PROGRAM pump_manager
VAR
	//Repeat for each pump?
	u_3112_b : motor_vfd;
	u_3112_b_pid : FB_BasicPID;
	u_3112_b_pid_error : UINT;
	u_3112_b_pid_output : REAL;
	u_3112_b_enable: BOOL;
	u_3112_b_idle_request: BOOL;
	u_3112_b_cip_request: BOOL;
	u_3112_b_manual_request: BOOL;
	u_3112_b_stop_request: BOOL;
	u_3112_b_intlk: BOOL;
	u_3112_b_maint_request: BOOL;
	u_3112_b_idle_speed_request: REAL;
	u_3112_b_setpoint_request: REAL;
	u_3112_b_cip_speed_request: REAL;
	u_3112_b_manual_speed_request: REAL;
	u_3112_b_maint_speed_request: REAL;
	
	u_3212_b : motor_vfd;
	u_3212_b_pid : FB_BasicPID;
	u_3212_b_pid_error : UINT;
	u_3212_b_enable: BOOL;
	u_3212_b_idle_request: BOOL;
	u_3212_b_cip_request: BOOL;
	u_3212_b_manual_request: BOOL;
	u_3212_b_stop_request: BOOL;
	u_3212_b_intlk: BOOL;
	u_3212_b_maint_request: BOOL;
	u_3212_b_idle_speed_request: REAL;
	u_3212_b_setpoint_request: REAL;
	u_3212_b_cip_speed_request: REAL;
	u_3212_b_manual_speed_request: REAL;
	u_3212_b_maint_speed_request: REAL;
	
	u_3312_b : motor_vfd;
	u_3312_b_pid : FB_BasicPID;
	u_3312_b_pid_error : UINT;
	u_3312_b_enable: BOOL;
	u_3312_b_idle_request: BOOL;
	u_3312_b_cip_request: BOOL;
	u_3312_b_manual_request: BOOL;
	u_3312_b_stop_request: BOOL;
	u_3312_b_intlk: BOOL;
	u_3312_b_maint_request: BOOL;
	u_3312_b_idle_speed_request: REAL;
	u_3312_b_speed_request: REAL;
	u_3312_b_cip_speed_request: REAL;
	u_3312_b_manual_speed_request: REAL;
	u_3312_b_maint_speed_request: REAL;
	
	u_3405_b : motor_vfd;
	u_3405_b_pid : FB_BasicPID;
	u_3405_b_pid_error : UINT;
	u_3405_b_enable: BOOL;
	u_3405_b_idle_request: BOOL;
	u_3405_b_cip_request: BOOL;
	u_3405_b_manual_request: BOOL;
	u_3405_b_stop_request: BOOL;
	u_3405_b_intlk: BOOL;
	u_3405_b_maint_request: BOOL;
	u_3405_b_idle_speed_request: REAL;
	u_3405_b_speed_request: REAL;
	u_3405_b_cip_speed_request: REAL;
	u_3405_b_manual_speed_request: REAL;
	u_3405_b_maint_speed_request: REAL;
	
	u_3160_b : motor_vfd;
	u_3160_b_pid : FB_BasicPID;
	u_3160_b_pid_error : UINT;
	u_3160_b_enable: BOOL;
	u_3160_b_idle_request: BOOL;
	u_3160_b_cip_request: BOOL;
	u_3160_b_manual_request: BOOL;
	u_3160_b_stop_request: BOOL;
	u_3160_b_intlk: BOOL;
	u_3160_b_maint_request: BOOL;
	u_3160_b_idle_speed_request: REAL;
	u_3160_b_speed_request: REAL;
	u_3160_b_cip_speed_request: REAL;
	u_3160_b_manual_speed_request: REAL;
	u_3160_b_maint_speed_request: REAL;
	
	u_3260_b : motor_vfd;
	u_3260_b_pid : FB_BasicPID;
	u_3260_b_pid_error : UINT;
	u_3260_b_enable: BOOL;
	u_3260_b_idle_request: BOOL;
	u_3260_b_cip_request: BOOL;
	u_3260_b_manual_request: BOOL;
	u_3260_b_stop_request: BOOL;
	u_3260_b_intlk: BOOL;
	u_3260_b_maint_request: BOOL;
	u_3260_b_idle_speed_request: REAL;
	u_3260_b_speed_request: REAL;
	u_3260_b_cip_speed_request: REAL;
	u_3260_b_manual_speed_request: REAL;
	u_3260_b_maint_speed_request: REAL;
	
	u_3360_b : motor_vfd;
	u_3360_b_pid : FB_BasicPID;
	u_3360_b_pid_error : UINT;
	u_3360_b_enable: BOOL;
	u_3360_b_idle_request: BOOL;
	u_3360_b_cip_request: BOOL;
	u_3360_b_manual_request: BOOL;
	u_3360_b_stop_request: BOOL;
	u_3360_b_intlk: BOOL;
	u_3360_b_maint_request: BOOL;
	u_3360_b_idle_speed_request: REAL;
	u_3360_b_speed_request: REAL;
	u_3360_b_cip_speed_request: REAL;
	u_3360_b_manual_speed_request: REAL;
	u_3360_b_maint_speed_request: REAL;
	
	
	gen_alm_active: BOOL;
	ed_routine_idle: BOOL;
	ed_routine_cip: BOOL;
	//ed_routine_manual: BOOL;
	ed_routine_maint: BOOL;
	
	u_3370_b : motor_vfd;
	u_3370_b_pid : FB_BasicPID;
	u_3370_b_pid_error : UINT;
	u_3370_b_enable: BOOL;
	u_3370_b_idle_request: BOOL;
	u_3370_b_cip_request: BOOL;
	u_3370_b_manual_request: BOOL;
	u_3370_b_stop_request: BOOL;
	u_3370_b_intlk: BOOL;
	u_3370_b_maint_request: BOOL;
	u_3370_b_idle_speed_request: REAL;
	u_3370_b_speed_request: REAL;
	u_3370_b_cip_speed_request: REAL;
	u_3370_b_manual_speed_request: REAL;
	u_3370_b_maint_speed_request: REAL;
	u_3312_b_setpoint_request: REAL;
	u_3405_b_setpoint_request: REAL;
	
	u_3112_b_pid_reset: BOOL;
	u_3112_b_ons: R_TRIG;
	u_3312_b_pid_reset: BOOL;
	u_3312_b_ons: R_TRIG;
	u_3212_b_ons: R_TRIG;
	u_3212_b_pid_reset: BOOL;
	u_3405_b_ons: R_TRIG;
	u_3405_b_pid_reset: BOOL;
	u_3370_b_setpoint_request: REAL;
	u_3370_b_ons: R_TRIG;
	u_3370_b_pid_reset: BOOL;
	u_3112_b_speed_request: REAL;
	u_3212_b_speed_request: REAL;
END_VAR
VAR // added by the converter: edge detectors and wires of the graphical bodies
    _w1, _w2, _w3, _w4, _w5, _w6, _w7, _w8, _w9, _w10, _w11, _w12, _w13, _w14, _w15, _w16, _w17, _w18, _w19, _w20, _w21, _w22, _w23, _w24, _w25, _w26, _w27, _w28 : BOOL;
END_VAR

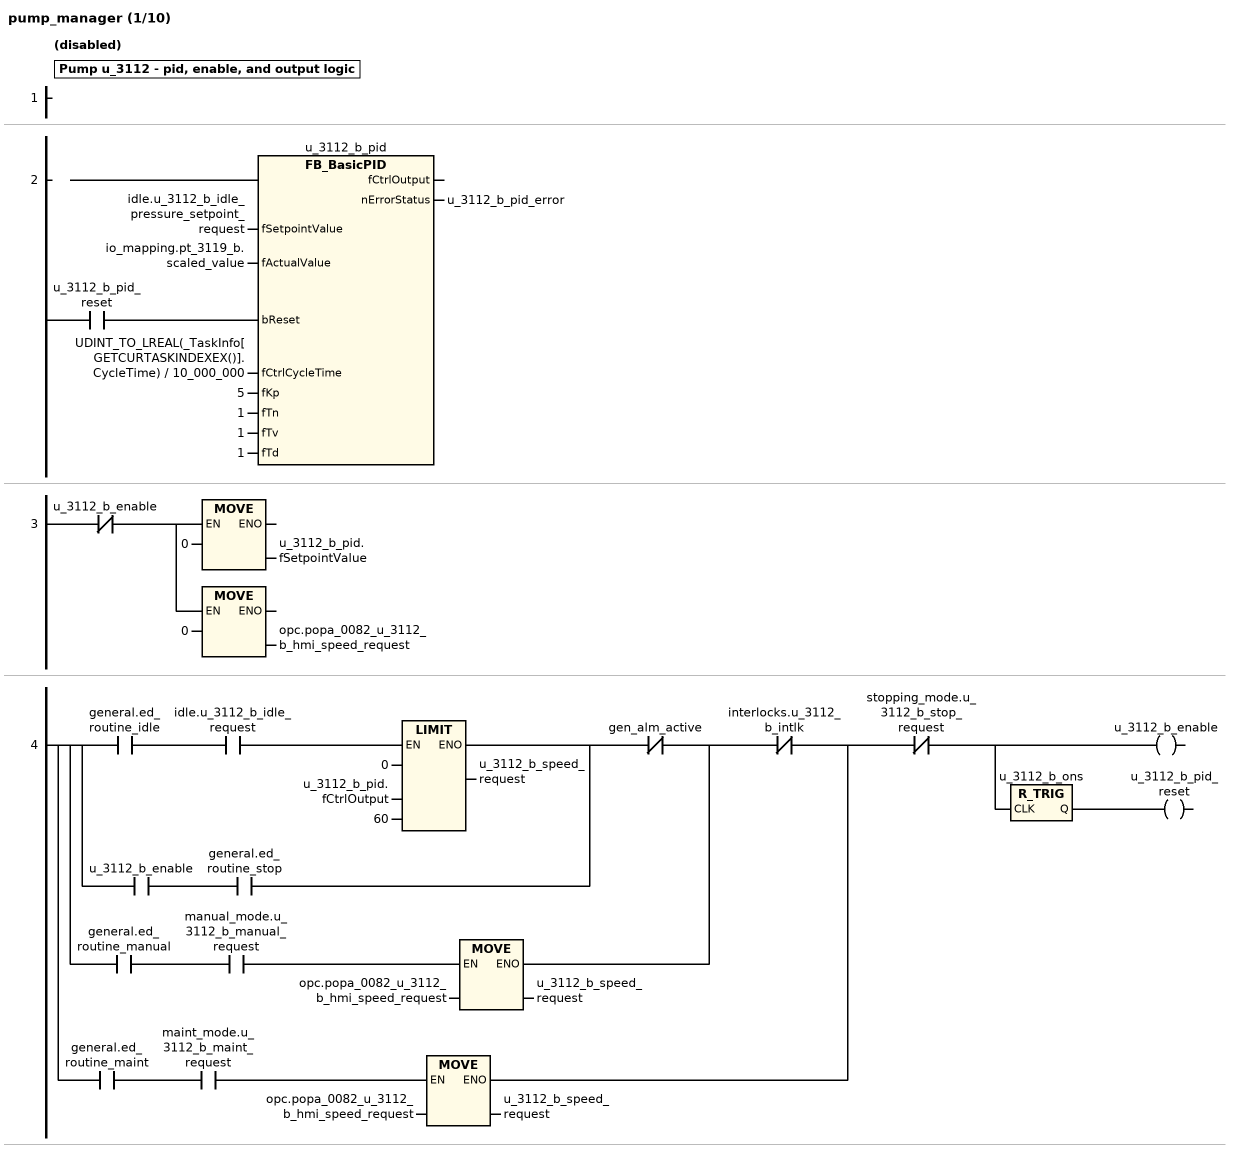
// NETWORK 1 (disabled)
// label: Pump u_3112 - pid, enable, and output logic

// NETWORK 2
u_3112_b_pid(
    fSetpointValue := idle.u_3112_b_idle_pressure_setpoint_request,
    fActualValue := io_mapping.pt_3119_b.scaled_value,
    bReset := u_3112_b_pid_reset,
    fCtrlCycleTime := UDINT_TO_LREAL(_TaskInfo[GETCURTASKINDEXEX()].CycleTime) / 10_000_000,
    fKp := 5,
    fTn := 1,
    fTv := 1,
    fTd := 1,
    nErrorStatus => u_3112_b_pid_error); // FB_BasicPID

// NETWORK 3
_w1 := NOT u_3112_b_enable;
IF _w1 THEN u_3112_b_pid.fSetpointValue := 0; END_IF
IF _w1 THEN opc.popa_0082_u_3112_b_hmi_speed_request := 0; END_IF

// NETWORK 4
_w2 := general.ed_routine_idle AND idle.u_3112_b_idle_request;
IF _w2 THEN u_3112_b_speed_request := LIMIT(0, u_3112_b_pid.fCtrlOutput, 60); END_IF
_w3 := general.ed_routine_manual AND manual_mode.u_3112_b_manual_request;
IF _w3 THEN u_3112_b_speed_request := opc.popa_0082_u_3112_b_hmi_speed_request; END_IF
_w4 := general.ed_routine_maint AND maint_mode.u_3112_b_maint_request;
IF _w4 THEN u_3112_b_speed_request := opc.popa_0082_u_3112_b_hmi_speed_request; END_IF
_w5 := (((_w2 OR u_3112_b_enable AND general.ed_routine_stop) AND NOT gen_alm_active OR _w3) AND NOT interlocks.u_3112_b_intlk OR _w4) AND NOT stopping_mode.u_3112_b_stop_request;
u_3112_b_enable := _w5;
u_3112_b_ons(CLK := _w5); // R_TRIG
u_3112_b_pid_reset := u_3112_b_ons.Q;

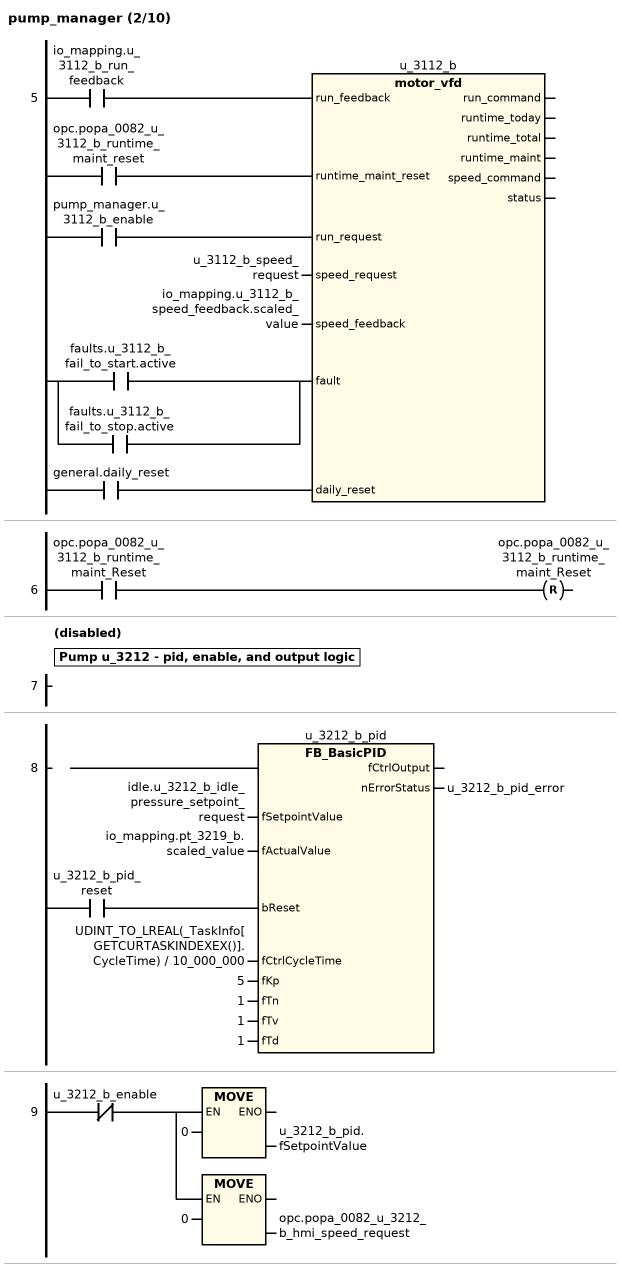
// NETWORK 5
u_3112_b(
    run_feedback := io_mapping.u_3112_b_run_feedback,
    runtime_maint_reset := opc.popa_0082_u_3112_b_runtime_maint_reset,
    run_request := pump_manager.u_3112_b_enable,
    speed_request := u_3112_b_speed_request,
    speed_feedback := io_mapping.u_3112_b_speed_feedback.scaled_value,
    fault := faults.u_3112_b_fail_to_start.active OR faults.u_3112_b_fail_to_stop.active,
    daily_reset := general.daily_reset); // motor_vfd

// NETWORK 6
opc.popa_0082_u_3112_b_runtime_maint_Reset R= opc.popa_0082_u_3112_b_runtime_maint_Reset;

// NETWORK 7 (disabled)
// label: Pump u_3212 - pid, enable, and output logic

// NETWORK 8
u_3212_b_pid(
    fSetpointValue := idle.u_3212_b_idle_pressure_setpoint_request,
    fActualValue := io_mapping.pt_3219_b.scaled_value,
    bReset := u_3212_b_pid_reset,
    fCtrlCycleTime := UDINT_TO_LREAL(_TaskInfo[GETCURTASKINDEXEX()].CycleTime) / 10_000_000,
    fKp := 5,
    fTn := 1,
    fTv := 1,
    fTd := 1,
    nErrorStatus => u_3212_b_pid_error); // FB_BasicPID

// NETWORK 9
_w6 := NOT u_3212_b_enable;
IF _w6 THEN u_3212_b_pid.fSetpointValue := 0; END_IF
IF _w6 THEN opc.popa_0082_u_3212_b_hmi_speed_request := 0; END_IF

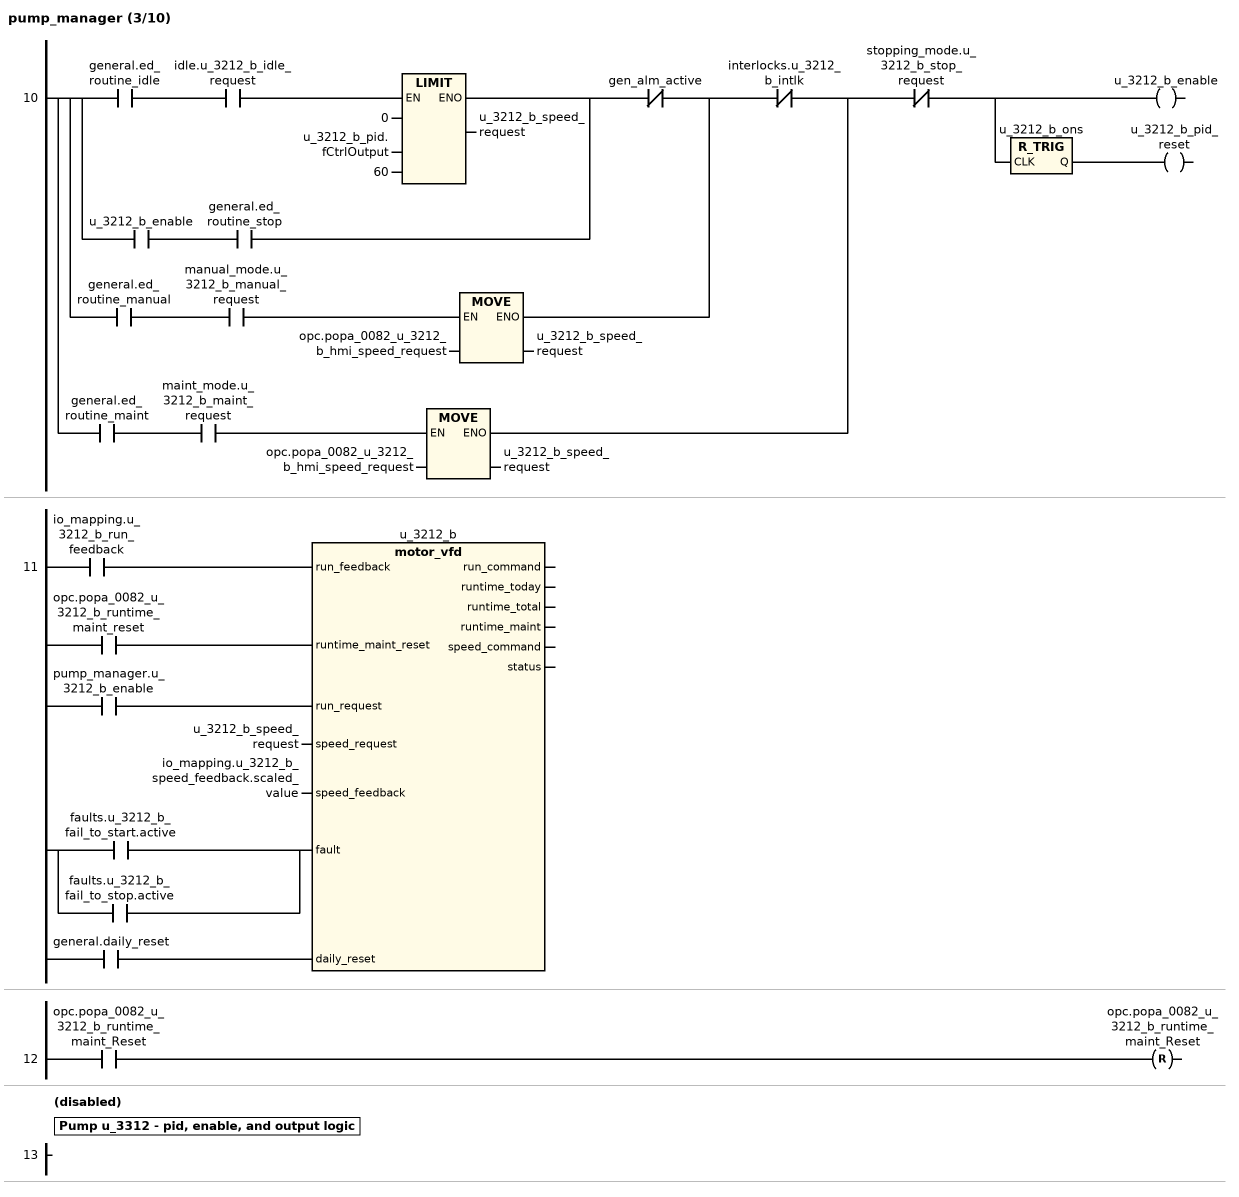
// NETWORK 10
_w7 := general.ed_routine_idle AND idle.u_3212_b_idle_request;
IF _w7 THEN u_3212_b_speed_request := LIMIT(0, u_3212_b_pid.fCtrlOutput, 60); END_IF
_w8 := general.ed_routine_manual AND manual_mode.u_3212_b_manual_request;
IF _w8 THEN u_3212_b_speed_request := opc.popa_0082_u_3212_b_hmi_speed_request; END_IF
_w9 := general.ed_routine_maint AND maint_mode.u_3212_b_maint_request;
IF _w9 THEN u_3212_b_speed_request := opc.popa_0082_u_3212_b_hmi_speed_request; END_IF
_w10 := (((_w7 OR u_3212_b_enable AND general.ed_routine_stop) AND NOT gen_alm_active OR _w8) AND NOT interlocks.u_3212_b_intlk OR _w9) AND NOT stopping_mode.u_3212_b_stop_request;
u_3212_b_enable := _w10;
u_3212_b_ons(CLK := _w10); // R_TRIG
u_3212_b_pid_reset := u_3212_b_ons.Q;

// NETWORK 11
u_3212_b(
    run_feedback := io_mapping.u_3212_b_run_feedback,
    runtime_maint_reset := opc.popa_0082_u_3212_b_runtime_maint_reset,
    run_request := pump_manager.u_3212_b_enable,
    speed_request := u_3212_b_speed_request,
    speed_feedback := io_mapping.u_3212_b_speed_feedback.scaled_value,
    fault := faults.u_3212_b_fail_to_start.active OR faults.u_3212_b_fail_to_stop.active,
    daily_reset := general.daily_reset); // motor_vfd

// NETWORK 12
opc.popa_0082_u_3212_b_runtime_maint_Reset R= opc.popa_0082_u_3212_b_runtime_maint_Reset;

// NETWORK 13 (disabled)
// label: Pump u_3312 - pid, enable, and output logic

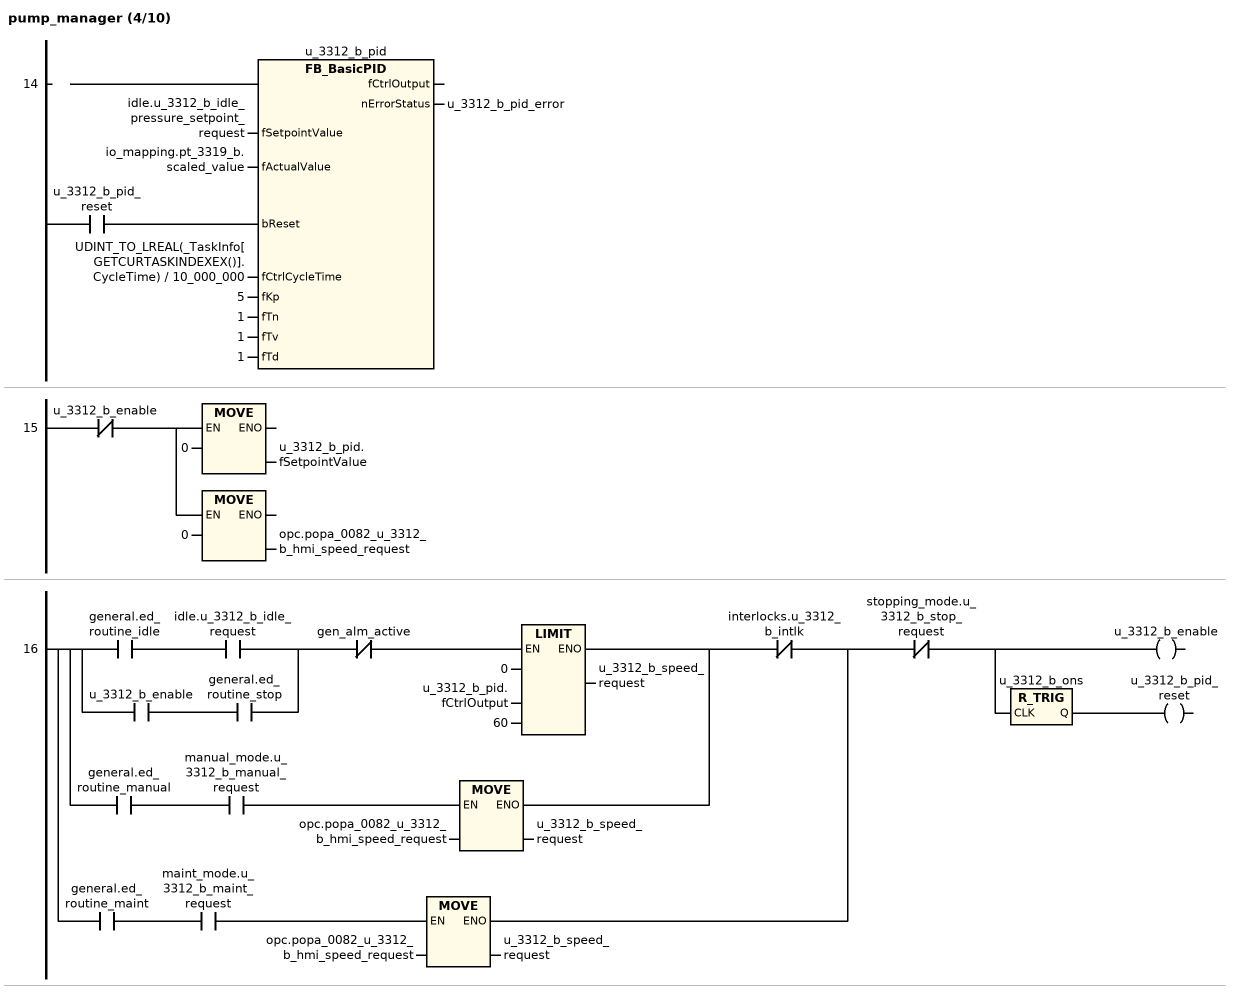
// NETWORK 14
u_3312_b_pid(
    fSetpointValue := idle.u_3312_b_idle_pressure_setpoint_request,
    fActualValue := io_mapping.pt_3319_b.scaled_value,
    bReset := u_3312_b_pid_reset,
    fCtrlCycleTime := UDINT_TO_LREAL(_TaskInfo[GETCURTASKINDEXEX()].CycleTime) / 10_000_000,
    fKp := 5,
    fTn := 1,
    fTv := 1,
    fTd := 1,
    nErrorStatus => u_3312_b_pid_error); // FB_BasicPID

// NETWORK 15
_w11 := NOT u_3312_b_enable;
IF _w11 THEN u_3312_b_pid.fSetpointValue := 0; END_IF
IF _w11 THEN opc.popa_0082_u_3312_b_hmi_speed_request := 0; END_IF

// NETWORK 16
_w12 := (general.ed_routine_idle AND idle.u_3312_b_idle_request OR u_3312_b_enable AND general.ed_routine_stop) AND NOT gen_alm_active;
IF _w12 THEN u_3312_b_speed_request := LIMIT(0, u_3312_b_pid.fCtrlOutput, 60); END_IF
_w13 := general.ed_routine_manual AND manual_mode.u_3312_b_manual_request;
IF _w13 THEN u_3312_b_speed_request := opc.popa_0082_u_3312_b_hmi_speed_request; END_IF
_w14 := general.ed_routine_maint AND maint_mode.u_3312_b_maint_request;
IF _w14 THEN u_3312_b_speed_request := opc.popa_0082_u_3312_b_hmi_speed_request; END_IF
_w15 := ((_w12 OR _w13) AND NOT interlocks.u_3312_b_intlk OR _w14) AND NOT stopping_mode.u_3312_b_stop_request;
u_3312_b_enable := _w15;
u_3312_b_ons(CLK := _w15); // R_TRIG
u_3312_b_pid_reset := u_3312_b_ons.Q;

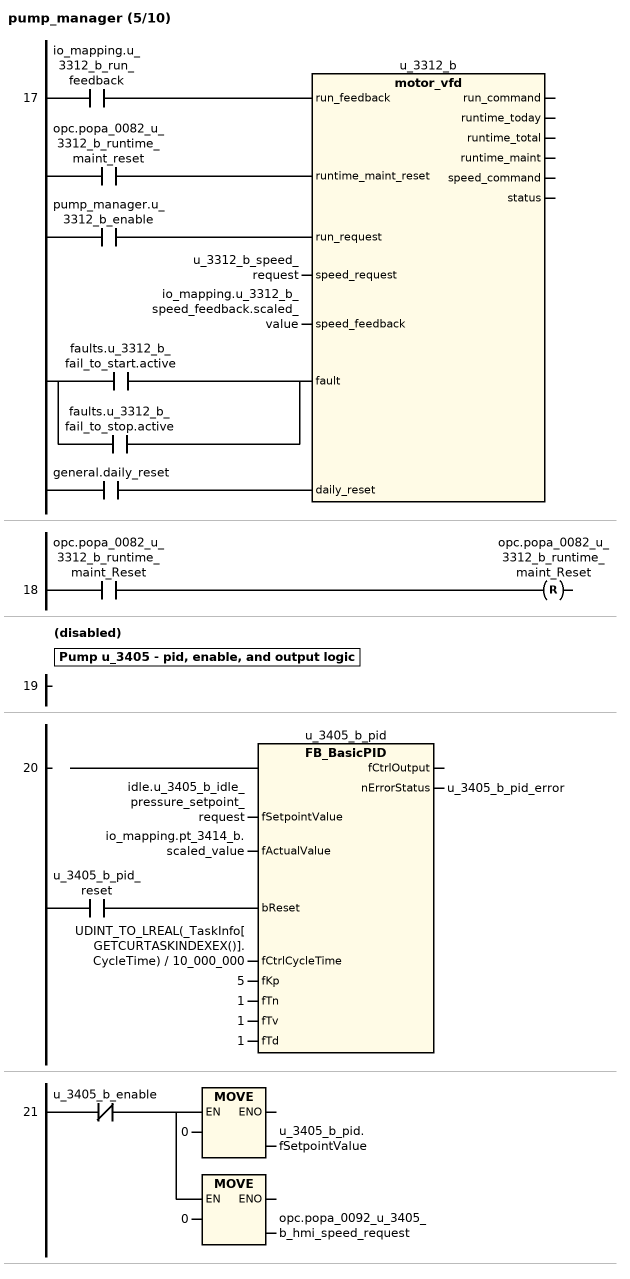
// NETWORK 17
u_3312_b(
    run_feedback := io_mapping.u_3312_b_run_feedback,
    runtime_maint_reset := opc.popa_0082_u_3312_b_runtime_maint_reset,
    run_request := pump_manager.u_3312_b_enable,
    speed_request := u_3312_b_speed_request,
    speed_feedback := io_mapping.u_3312_b_speed_feedback.scaled_value,
    fault := faults.u_3312_b_fail_to_start.active OR faults.u_3312_b_fail_to_stop.active,
    daily_reset := general.daily_reset); // motor_vfd

// NETWORK 18
opc.popa_0082_u_3312_b_runtime_maint_Reset R= opc.popa_0082_u_3312_b_runtime_maint_Reset;

// NETWORK 19 (disabled)
// label: Pump u_3405 - pid, enable, and output logic

// NETWORK 20
u_3405_b_pid(
    fSetpointValue := idle.u_3405_b_idle_pressure_setpoint_request,
    fActualValue := io_mapping.pt_3414_b.scaled_value,
    bReset := u_3405_b_pid_reset,
    fCtrlCycleTime := UDINT_TO_LREAL(_TaskInfo[GETCURTASKINDEXEX()].CycleTime) / 10_000_000,
    fKp := 5,
    fTn := 1,
    fTv := 1,
    fTd := 1,
    nErrorStatus => u_3405_b_pid_error); // FB_BasicPID

// NETWORK 21
_w16 := NOT u_3405_b_enable;
IF _w16 THEN u_3405_b_pid.fSetpointValue := 0; END_IF
IF _w16 THEN opc.popa_0092_u_3405_b_hmi_speed_request := 0; END_IF

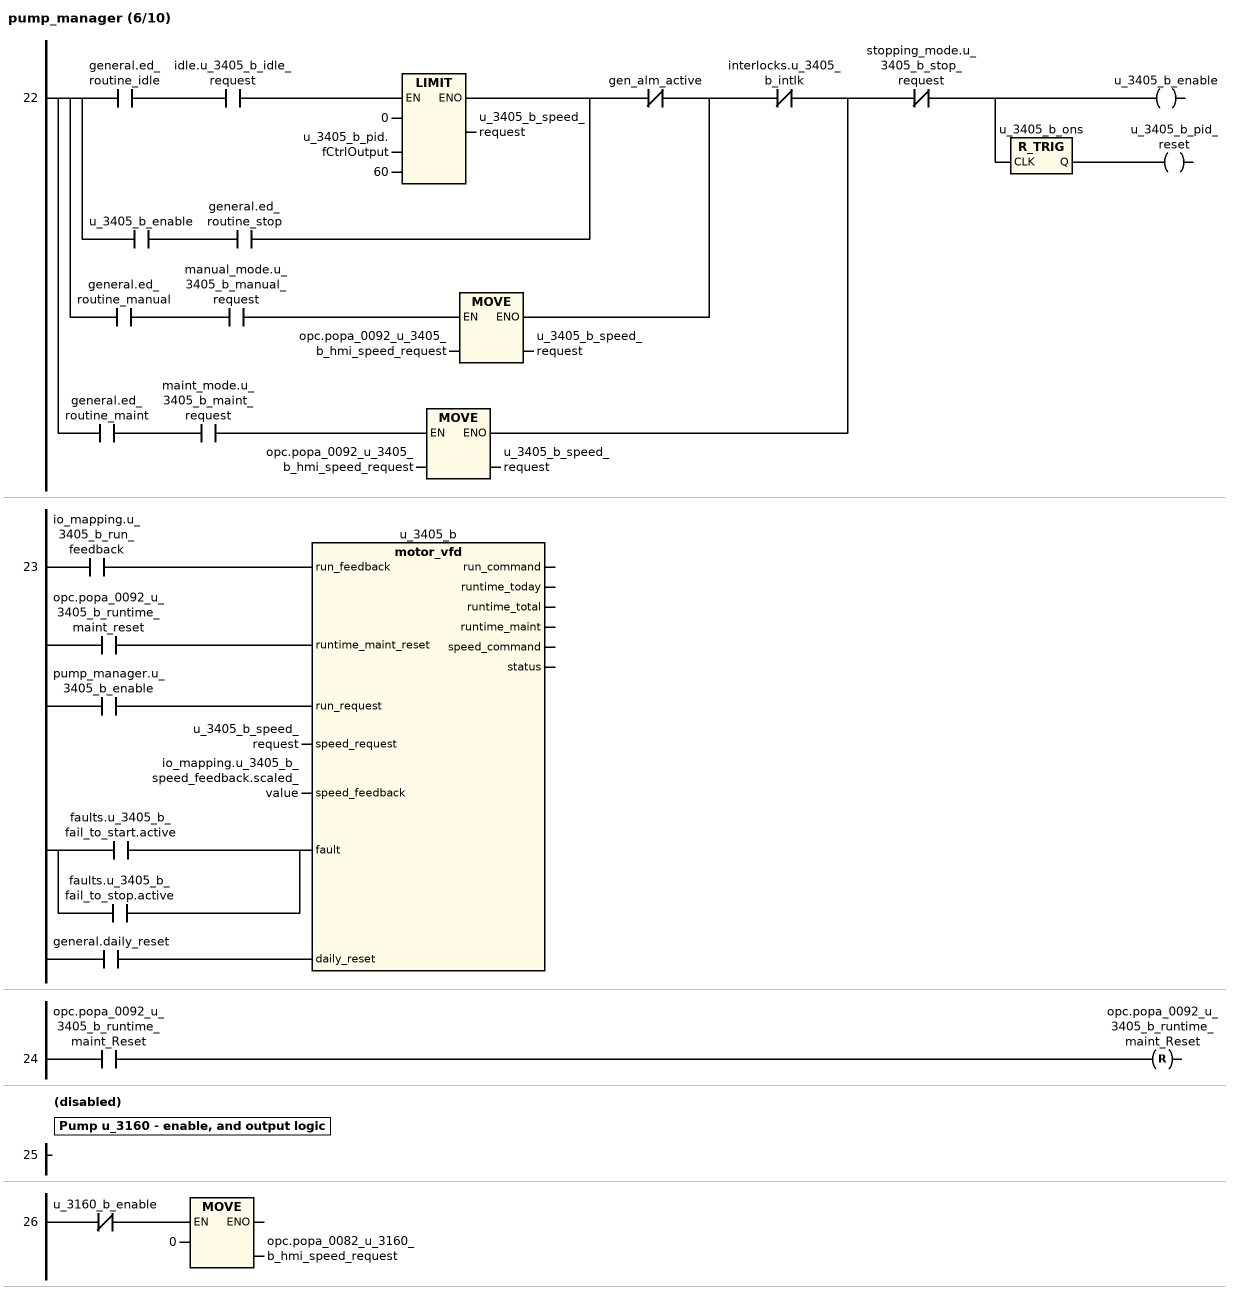
// NETWORK 22
_w17 := general.ed_routine_idle AND idle.u_3405_b_idle_request;
IF _w17 THEN u_3405_b_speed_request := LIMIT(0, u_3405_b_pid.fCtrlOutput, 60); END_IF
_w18 := general.ed_routine_manual AND manual_mode.u_3405_b_manual_request;
IF _w18 THEN u_3405_b_speed_request := opc.popa_0092_u_3405_b_hmi_speed_request; END_IF
_w19 := general.ed_routine_maint AND maint_mode.u_3405_b_maint_request;
IF _w19 THEN u_3405_b_speed_request := opc.popa_0092_u_3405_b_hmi_speed_request; END_IF
_w20 := (((_w17 OR u_3405_b_enable AND general.ed_routine_stop) AND NOT gen_alm_active OR _w18) AND NOT interlocks.u_3405_b_intlk OR _w19) AND NOT stopping_mode.u_3405_b_stop_request;
u_3405_b_enable := _w20;
u_3405_b_ons(CLK := _w20); // R_TRIG
u_3405_b_pid_reset := u_3405_b_ons.Q;

// NETWORK 23
u_3405_b(
    run_feedback := io_mapping.u_3405_b_run_feedback,
    runtime_maint_reset := opc.popa_0092_u_3405_b_runtime_maint_reset,
    run_request := pump_manager.u_3405_b_enable,
    speed_request := u_3405_b_speed_request,
    speed_feedback := io_mapping.u_3405_b_speed_feedback.scaled_value,
    fault := faults.u_3405_b_fail_to_start.active OR faults.u_3405_b_fail_to_stop.active,
    daily_reset := general.daily_reset); // motor_vfd

// NETWORK 24
opc.popa_0092_u_3405_b_runtime_maint_Reset R= opc.popa_0092_u_3405_b_runtime_maint_Reset;

// NETWORK 25 (disabled)
// label: Pump u_3160 - enable, and output logic

// NETWORK 26
IF NOT u_3160_b_enable THEN opc.popa_0082_u_3160_b_hmi_speed_request := 0; END_IF

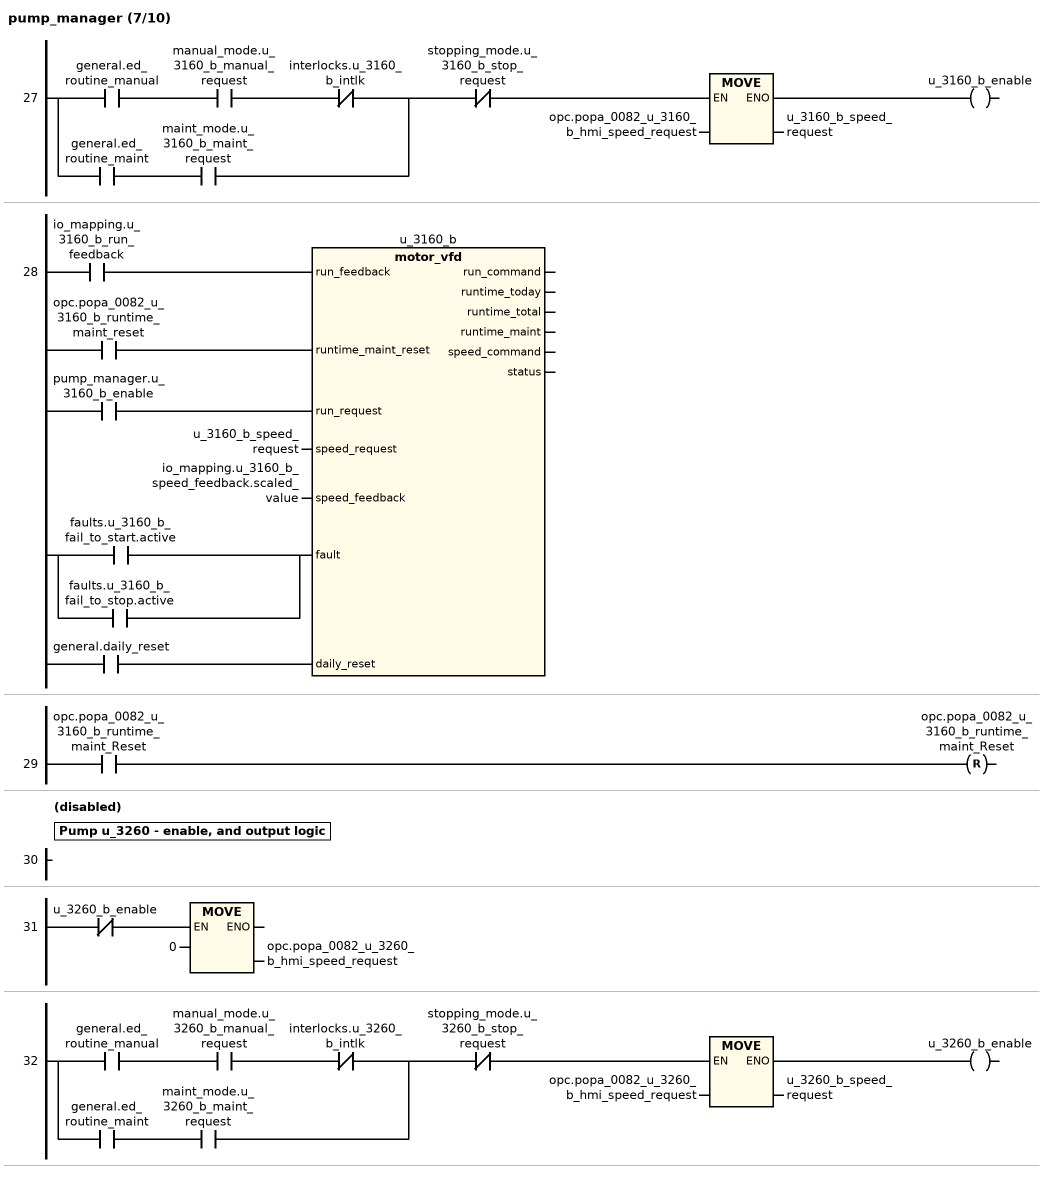
// NETWORK 27
_w21 := (general.ed_routine_manual AND manual_mode.u_3160_b_manual_request AND NOT interlocks.u_3160_b_intlk OR general.ed_routine_maint AND maint_mode.u_3160_b_maint_request) AND NOT stopping_mode.u_3160_b_stop_request;
IF _w21 THEN u_3160_b_speed_request := opc.popa_0082_u_3160_b_hmi_speed_request; END_IF
u_3160_b_enable := _w21;

// NETWORK 28
u_3160_b(
    run_feedback := io_mapping.u_3160_b_run_feedback,
    runtime_maint_reset := opc.popa_0082_u_3160_b_runtime_maint_reset,
    run_request := pump_manager.u_3160_b_enable,
    speed_request := u_3160_b_speed_request,
    speed_feedback := io_mapping.u_3160_b_speed_feedback.scaled_value,
    fault := faults.u_3160_b_fail_to_start.active OR faults.u_3160_b_fail_to_stop.active,
    daily_reset := general.daily_reset); // motor_vfd

// NETWORK 29
opc.popa_0082_u_3160_b_runtime_maint_Reset R= opc.popa_0082_u_3160_b_runtime_maint_Reset;

// NETWORK 30 (disabled)
// label: Pump u_3260 - enable, and output logic

// NETWORK 31
IF NOT u_3260_b_enable THEN opc.popa_0082_u_3260_b_hmi_speed_request := 0; END_IF

// NETWORK 32
_w22 := (general.ed_routine_manual AND manual_mode.u_3260_b_manual_request AND NOT interlocks.u_3260_b_intlk OR general.ed_routine_maint AND maint_mode.u_3260_b_maint_request) AND NOT stopping_mode.u_3260_b_stop_request;
IF _w22 THEN u_3260_b_speed_request := opc.popa_0082_u_3260_b_hmi_speed_request; END_IF
u_3260_b_enable := _w22;

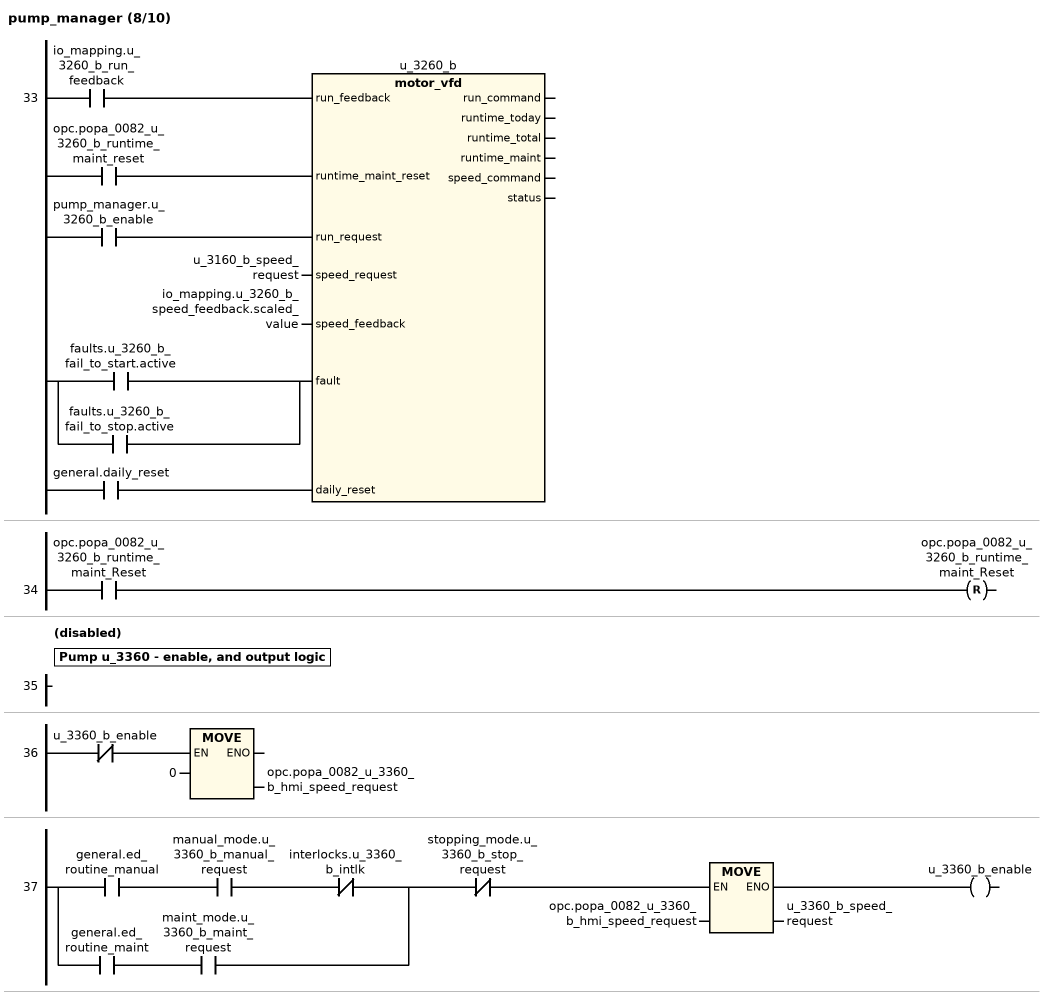
// NETWORK 33
u_3260_b(
    run_feedback := io_mapping.u_3260_b_run_feedback,
    runtime_maint_reset := opc.popa_0082_u_3260_b_runtime_maint_reset,
    run_request := pump_manager.u_3260_b_enable,
    speed_request := u_3160_b_speed_request,
    speed_feedback := io_mapping.u_3260_b_speed_feedback.scaled_value,
    fault := faults.u_3260_b_fail_to_start.active OR faults.u_3260_b_fail_to_stop.active,
    daily_reset := general.daily_reset); // motor_vfd

// NETWORK 34
opc.popa_0082_u_3260_b_runtime_maint_Reset R= opc.popa_0082_u_3260_b_runtime_maint_Reset;

// NETWORK 35 (disabled)
// label: Pump u_3360 - enable, and output logic

// NETWORK 36
IF NOT u_3360_b_enable THEN opc.popa_0082_u_3360_b_hmi_speed_request := 0; END_IF

// NETWORK 37
_w23 := (general.ed_routine_manual AND manual_mode.u_3360_b_manual_request AND NOT interlocks.u_3360_b_intlk OR general.ed_routine_maint AND maint_mode.u_3360_b_maint_request) AND NOT stopping_mode.u_3360_b_stop_request;
IF _w23 THEN u_3360_b_speed_request := opc.popa_0082_u_3360_b_hmi_speed_request; END_IF
u_3360_b_enable := _w23;

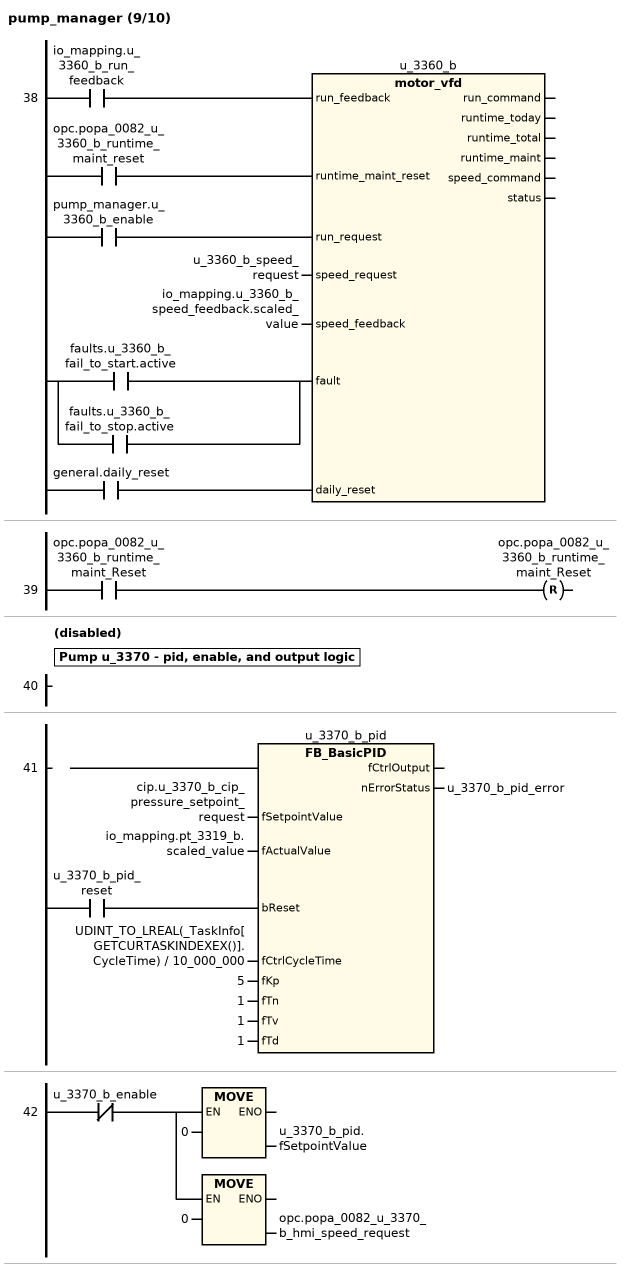
// NETWORK 38
u_3360_b(
    run_feedback := io_mapping.u_3360_b_run_feedback,
    runtime_maint_reset := opc.popa_0082_u_3360_b_runtime_maint_reset,
    run_request := pump_manager.u_3360_b_enable,
    speed_request := u_3360_b_speed_request,
    speed_feedback := io_mapping.u_3360_b_speed_feedback.scaled_value,
    fault := faults.u_3360_b_fail_to_start.active OR faults.u_3360_b_fail_to_stop.active,
    daily_reset := general.daily_reset); // motor_vfd

// NETWORK 39
opc.popa_0082_u_3360_b_runtime_maint_Reset R= opc.popa_0082_u_3360_b_runtime_maint_Reset;

// NETWORK 40 (disabled)
// label: Pump u_3370 - pid, enable, and output logic

// NETWORK 41
u_3370_b_pid(
    fSetpointValue := cip.u_3370_b_cip_pressure_setpoint_request,
    fActualValue := io_mapping.pt_3319_b.scaled_value,
    bReset := u_3370_b_pid_reset,
    fCtrlCycleTime := UDINT_TO_LREAL(_TaskInfo[GETCURTASKINDEXEX()].CycleTime) / 10_000_000,
    fKp := 5,
    fTn := 1,
    fTv := 1,
    fTd := 1,
    nErrorStatus => u_3370_b_pid_error); // FB_BasicPID

// NETWORK 42
_w24 := NOT u_3370_b_enable;
IF _w24 THEN u_3370_b_pid.fSetpointValue := 0; END_IF
IF _w24 THEN opc.popa_0082_u_3370_b_hmi_speed_request := 0; END_IF

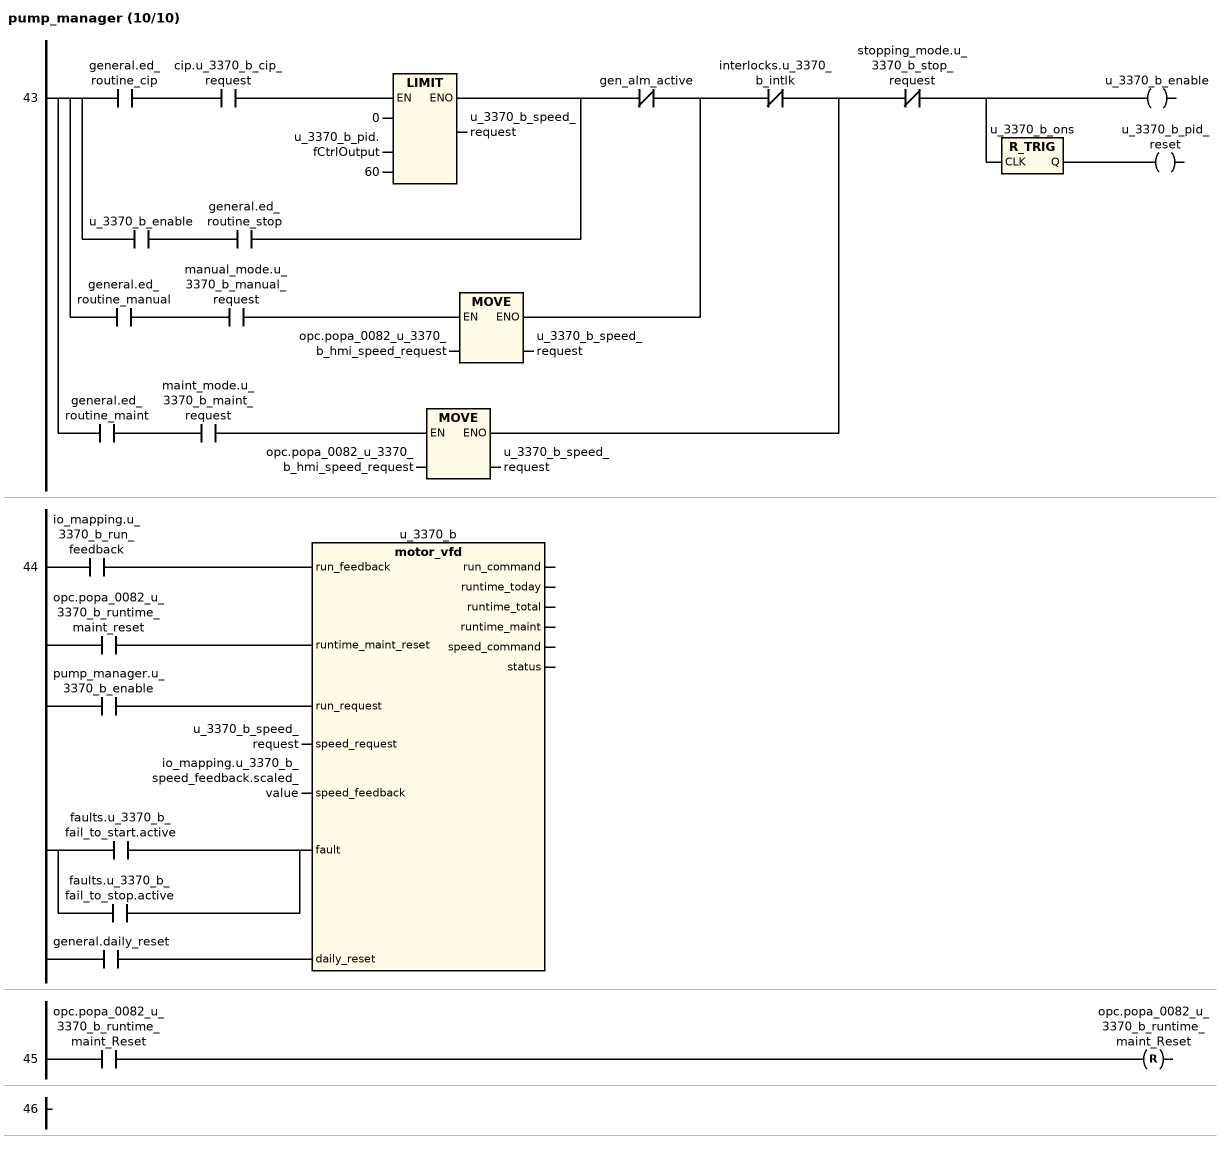
// NETWORK 43
_w25 := general.ed_routine_cip AND cip.u_3370_b_cip_request;
IF _w25 THEN u_3370_b_speed_request := LIMIT(0, u_3370_b_pid.fCtrlOutput, 60); END_IF
_w26 := general.ed_routine_manual AND manual_mode.u_3370_b_manual_request;
IF _w26 THEN u_3370_b_speed_request := opc.popa_0082_u_3370_b_hmi_speed_request; END_IF
_w27 := general.ed_routine_maint AND maint_mode.u_3370_b_maint_request;
IF _w27 THEN u_3370_b_speed_request := opc.popa_0082_u_3370_b_hmi_speed_request; END_IF
_w28 := (((_w25 OR u_3370_b_enable AND general.ed_routine_stop) AND NOT gen_alm_active OR _w26) AND NOT interlocks.u_3370_b_intlk OR _w27) AND NOT stopping_mode.u_3370_b_stop_request;
u_3370_b_enable := _w28;
u_3370_b_ons(CLK := _w28); // R_TRIG
u_3370_b_pid_reset := u_3370_b_ons.Q;

// NETWORK 44
u_3370_b(
    run_feedback := io_mapping.u_3370_b_run_feedback,
    runtime_maint_reset := opc.popa_0082_u_3370_b_runtime_maint_reset,
    run_request := pump_manager.u_3370_b_enable,
    speed_request := u_3370_b_speed_request,
    speed_feedback := io_mapping.u_3370_b_speed_feedback.scaled_value,
    fault := faults.u_3370_b_fail_to_start.active OR faults.u_3370_b_fail_to_stop.active,
    daily_reset := general.daily_reset); // motor_vfd

// NETWORK 45
opc.popa_0082_u_3370_b_runtime_maint_Reset R= opc.popa_0082_u_3370_b_runtime_maint_Reset;

// NETWORK 46

END_PROGRAM

(* stored: Version 1.1.0.1, ProductVersion 3.1.4024.15
   POU pump_manager: Id {3b5ad67c-a464-4c74-9317-fc4708b2e954}, SpecialFunc None *)
